FUNCTION_BLOCK cvtColor (* openCV color conversion *)
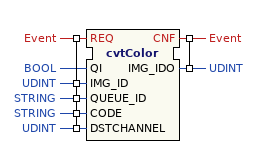
  EVENT_INPUT
    REQ WITH IMG_ID, QUEUE_ID, CODE, DSTCHANNEL;
  END_EVENT
  EVENT_OUTPUT
    CNF WITH IMG_IDO;
  END_EVENT
  VAR_INPUT
    QI : BOOL;
    IMG_ID : UDINT;
    QUEUE_ID : STRING;
    CODE : STRING;
    DSTCHANNEL : UDINT;
  END_VAR
  VAR_OUTPUT
    IMG_IDO : UDINT;
  END_VAR
END_FUNCTION_BLOCK
